TYPE ST_SICK :
STRUCT
END_STRUCT
END_TYPE

(* stored: Version 1.1.0.1, ProductVersion 3.1.4022.11
   DUT ST_SICK: Id {f2725782-64b9-4ba1-bbc4-9cb237499b94} *)
